SUBAPPLICATION Uebung_002a5b (* DigitalInput_I1-3 mit OR auf DigitalOutput_Q1-3 *)
  (* Standard: 61499-2; Description: Copyright (c) 2023 Meisterschulen am Ostbahnhof This program and the accompanying materials are made available under the terms of the Eclipse Public License 2.0 which is available at https://www.eclipse.org/legal/epl-2.0/ SPDX-License-Identifier: EPL-2.0 *)
  (* Version 1.0, 2023-10-23, Franz Höpfinger, Meisterschulen am Ostbahnhof *)
  PACKAGE Uebungen;
  IMPORT logiBUS::io::DI::logiBUS_DI::Input_I1;
  IMPORT logiBUS::io::DI::logiBUS_DI::Input_I2;
  IMPORT logiBUS::io::DI::logiBUS_DI::Input_I3;
  IMPORT logiBUS::io::DQ::logiBUS_DO::Output_Q1;
  IMPORT logiBUS::io::DQ::logiBUS_DO::Output_Q2;
  IMPORT logiBUS::io::DQ::logiBUS_DO::Output_Q3;
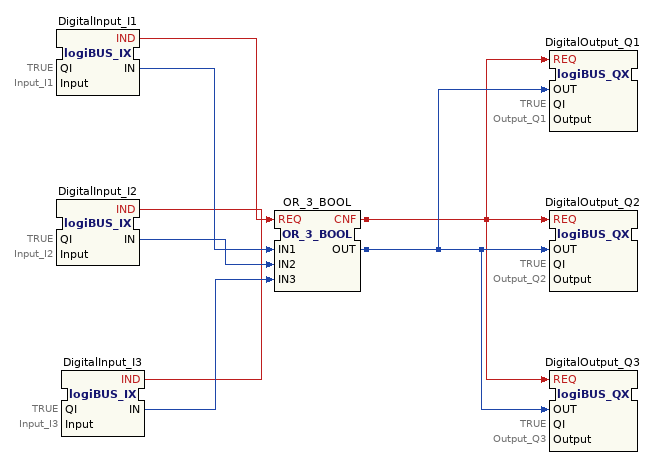
  FBS
    DigitalOutput_Q1 : logiBUS::io::DQ::logiBUS_QX(QI := TRUE, Output := Output_Q1);
    DigitalInput_I1 : logiBUS::io::DI::logiBUS_IX(QI := TRUE, Input := Input_I1);
    DigitalInput_I2 : logiBUS::io::DI::logiBUS_IX(QI := TRUE, Input := Input_I2);
    DigitalInput_I3 : logiBUS::io::DI::logiBUS_IX(QI := TRUE, Input := Input_I3);
    DigitalOutput_Q2 : logiBUS::io::DQ::logiBUS_QX(QI := TRUE, Output := Output_Q2);
    DigitalOutput_Q3 : logiBUS::io::DQ::logiBUS_QX(QI := TRUE, Output := Output_Q3);
    OR_3_BOOL : iec61131::bitwiseOperators::OR_3_BOOL;
  END_FBS
  EVENT_CONNECTIONS
    DigitalInput_I1.IND TO OR_3_BOOL.REQ;
    DigitalInput_I2.IND TO OR_3_BOOL.REQ;
    DigitalInput_I3.IND TO OR_3_BOOL.REQ;
    OR_3_BOOL.CNF TO DigitalOutput_Q1.REQ;
    OR_3_BOOL.CNF TO DigitalOutput_Q2.REQ;
    OR_3_BOOL.CNF TO DigitalOutput_Q3.REQ;
  END_CONNECTIONS
  DATA_CONNECTIONS
    DigitalInput_I1.IN TO OR_3_BOOL.IN1;
    DigitalInput_I2.IN TO OR_3_BOOL.IN2;
    DigitalInput_I3.IN TO OR_3_BOOL.IN3;
    OR_3_BOOL.OUT TO DigitalOutput_Q1.OUT;
    OR_3_BOOL.OUT TO DigitalOutput_Q2.OUT;
    OR_3_BOOL.OUT TO DigitalOutput_Q3.OUT;
  END_CONNECTIONS
END_SUBAPPLICATION
